FUNCTION_BLOCK AL_TO_ALR (* Composite FB for converting AL (LWORD) adapter to ALR (LREAL) adapter — ⚠ BIT-REINTERPRETATION, NOT a numeric cast! A raw counter/analog value is misinterpreted as IEEE754 bits. See AD_TO_AR_TODO.md / AD_TO_AR_NUM for the safe two-stage (bit-string->int->real) alternative. *)
  (* Standard: 61499-2; Description: Copyright (c) 2026 HR Agrartechnik GmbH This program and the accompanying materials are made available under the terms of the Eclipse Public License 2.0 which is available at https://www.eclipse.org/legal/epl-2.0/ SPDX-License-Identifier: EPL-2.0 *)
  (* Version 1.0, 2026-02-17, Franz Höpfinger, HR Agrartechnik GmbH *)
  PACKAGE adapter::conversion::unidirectional;
  (* Documentation:
  AL_TO_ALR
   🇩🇪 Deutsch
   ⚠️ Achtung: Dieser Baustein wandelt LWORD nicht numerisch in LREAL um, sondern nutzt intern F_LWORD_TO_LREAL, was im FORTE-Kern für Bit-String-Quelltypen (BYTE/WORD/DWORD/LWORD) eine reine IEEE754-Bit-Reinterpretation ist — dieselbe Falle wie bei AD_TO_AR (DWORD→REAL), hier nur mit den 64-bit-Pendants LWORD/LREAL. Ein roher Zähler-/Analogwert würde dadurch NICHT in den entsprechenden REAL-Zahlenwert umgewandelt, sondern ergäbe eine bedeutungslose Zahl.
   AL_TO_ALR ist trotzdem korrekt, wenn AL_IN bereits ein Bitmuster ist, das als LREAL interpretiert werden soll (z. B. das Ergebnis eines F_LREAL_TO_LWORD).
   Für einen echten Zahlenwert: zweistufig über AL_TO_AULI (Bit-Reinterpretation LWORD→ULINT, hier gültig, da beide dieselbe 64-bit-Darstellung eines vorzeichenlosen Integers teilen) gefolgt von AULI_TO_ALR (echter numerischer Cast) — dasselbe Muster wie AD_TO_AR_NUM für den 32-bit-Fall.
   🇬🇧 English
   ⚠️ Warning: This block does not numerically convert LWORD to LREAL — it internally uses F_LWORD_TO_LREAL, which in the FORTE core is a pure IEEE754 bit-reinterpretation for bit-string source types (BYTE/WORD/DWORD/LWORD) — the same trap as AD_TO_AR (DWORD→REAL), here with the 64-bit counterparts LWORD/LREAL. A raw counter/analog value would NOT become the corresponding REAL number, but a meaningless value.
   AL_TO_ALR is still correct when AL_IN is already a bit pattern meant to be interpreted as LREAL (e.g. the result of an F_LREAL_TO_LWORD).
   For an actual numeric value: chain AL_TO_AULI (bit-reinterpretation LWORD→ULINT, valid here since both share the same 64-bit unsigned-integer representation) followed by AULI_TO_ALR (a real numeric cast) — the same pattern as AD_TO_AR_NUM for the 32-bit case.
  *)
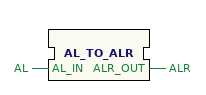
  SOCKETS
    AL_IN : adapter::types::unidirectional::AL; (* LWORD Adapter Input *)
  END_SOCKETS
  PLUGS
    ALR_OUT : adapter::types::unidirectional::ALR; (* LREAL Adapter Output *)
  END_PLUGS
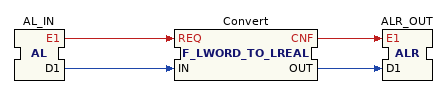
  FBS
    Convert : iec61131::conversion::F_LWORD_TO_LREAL;
  END_FBS
  EVENT_CONNECTIONS
    AL_IN.E1 TO Convert.REQ;
    Convert.CNF TO ALR_OUT.E1;
  END_CONNECTIONS
  DATA_CONNECTIONS
    AL_IN.D1 TO Convert.IN;
    Convert.OUT TO ALR_OUT.D1;
  END_CONNECTIONS
END_FUNCTION_BLOCK
